{attribute 'linkalways'} 
{attribute 'no_explicit_call' := 'This FB is a CLASS and must be accessed using methods or properties'}
{attribute 'enable_dynamic_creation'}
FUNCTION_BLOCK FINAL NE_LINT EXTENDS Node
VAR
	in1 : _LINT(0);
	in2 : _LINT(0);
	out : _BOOL(FALSE);
END_VAR

METHOD PUBLIC Clone : I_Node
VAR
	pNode : POINTER TO NE_LINT;
END_VAR
pNode := __NEW(NE_LINT);
Clone := pNode^;
END_METHOD

METHOD FB_init : BOOL
VAR_INPUT
	bInitRetains : BOOL; // if TRUE, the retain variables are initialized (warm start / cold start)
	bInCopyCode : BOOL;  // if TRUE, the instance afterwards gets moved into the copy code (online change)
END_VAR
AddInput('in1',THIS^.in1);
AddInput('in2',THIS^.in2);
AddOutput('out', THIS^.out);
END_METHOD

METHOD PROTECTED OnExecute
VAR
END_VAR
out.Value := in1.Value <> in2.Value;
END_METHOD

END_FUNCTION_BLOCK

(* stored: Version 1.1.0.1, ProductVersion 3.1.4024.15
   POU NE_LINT: Id {3a5f3387-7fd9-426a-b9f9-896d70b23b9a}, SpecialFunc None
   Folder Constructor: Id {606d0d41-061a-430d-85fc-a7d356db109c}
   Method Clone: Id {11014c87-456b-4a89-8d40-0b0b986c58af}
   Method FB_init: Id {f778421a-d182-462b-b0de-eff20d3bcf10}
   Method OnExecute: Id {3d3722b3-ea48-4f61-bb09-80de1f94aef9} *)
